// TIA Portal V20 export
TYPE "typeCmControlNodeSoftCamsideTapeAttachmentAxisY"
// stored: Namespace Unit1.Em4
   STRUCT
      Pos00_wait : "LER_typeSoftCamPosition";
      pos01_rightTapeGet : "LER_typeSoftCamPosition";
      pos02_leftTapeGet : "LER_typeSoftCamPosition";
      pos03_tape1Put : "LER_typeSoftCamPosition";
      pos04_tape2Put : "LER_typeSoftCamPosition";
      pos05_tape3Put : "LER_typeSoftCamPosition";
      pos06_tape4Put : "LER_typeSoftCamPosition";
      pos07_remainAttachLeft : "LER_typeSoftCamPosition";
      pos08_remainAttachRight : "LER_typeSoftCamPosition";
      pos09_noInterferenceZone : "LER_typeSoftCamPosition";
      pos10_posistion : "LER_typeSoftCamPosition";
      pos11_posistion : "LER_typeSoftCamPosition";
      pos12_posistion : "LER_typeSoftCamPosition";
      pos13_posistion : "LER_typeSoftCamPosition";
      pos14_posistion : "LER_typeSoftCamPosition";
      pos15_posistion : "LER_typeSoftCamPosition";
   END_STRUCT;
END_TYPE
